FUNCTION_BLOCK FB_JoystickInputScaling
VAR_INPUT
	bEnable 				: BOOL;
	nRawInput 				: INT;
	stJoystickInputScaling  : ST_JoystickInputScaling;
END_VAR
VAR_OUTPUT
	fNormalizedOutput 		: LREAL;
END_VAR
VAR
	fRawInput 				: LREAL;
	fTempInput 				: LREAL;
	fTempOutput 			: LREAL;
END_VAR

fRawInput := INT_TO_LREAL(nRawInput);

fTempInput := fRawInput - stJoystickInputScaling.fNeutralInputValue;

IF fTempInput > stJoystickInputScaling.fNeutralDeadband THEN
	fTempOutput := fTempInput/(stJoystickInputScaling.fMaxInputValue - stJoystickInputScaling.fNeutralInputValue);
ELSIF fTempInput < -stJoystickInputScaling.fNeutralDeadband THEN	
	fTempOutput := fTempInput/(stJoystickInputScaling.fNeutralInputValue - stJoystickInputScaling.fMinInputValue);
ELSE
	fTempOutput := 0.0;
END_IF

IF NOT(bEnable) THEN
	fNormalizedOutput := 0.0;
ELSE
	fNormalizedOutput := LIMIT(stJoystickInputScaling.fMinOutputValue, fTempOutput, stJoystickInputScaling.fMaxOutputValue);
END_IF

END_FUNCTION_BLOCK

(* stored: Version 1.1.0.1, ProductVersion 3.1.4024.11
   POU FB_JoystickInputScaling: Id {45abe8f1-3862-4b14-9ee2-cf88212f6af6}, SpecialFunc None *)
